FUNCTION_BLOCK T_RisingEdge
VAR
    R_TRIG1 : R_TRIG;
END_VAR

PROPERTY EdgeDetected : BOOL
GET
EdgeDetected := R_TRIG1.Q;
END_GET
END_PROPERTY

METHOD Test : BOOL
VAR_INPUT
    Value : BOOL;
END_VAR
R_TRIG1(CLK := Value);
Test := R_TRIG1.Q;
END_METHOD

END_FUNCTION_BLOCK

(* stored: Version 1.1.0.1, ProductVersion 3.1.4024.4
   POU T_RisingEdge: Id {59aed088-2301-02c0-044b-6e8c897b9b7e}, SpecialFunc None
   Property EdgeDetected: Id {c670d64f-39a9-0e02-36d1-2a2447c5caea}
   Get Get: Id {95fd47b6-9165-0ff6-2b79-9d0db693a8d1}
   Method Test: Id {842f4957-e5af-0186-0606-af3122602df9} *)
